(* PLC project OOP_Curso, Beckhoff Automation GmbH TwinCAT PLC Control 3.5.13.21 *)
(* stored: creationDateTime 2023-04-23T11:42:48.8573622, modificationDateTime 2023-04-23T11:42:48.8641947 *)

INTERFACE I_Employee
METHOD GetFullName : STRING
VAR_INPUT
END_VAR
END_METHOD
METHOD GetMonthlySalary : LREAL
VAR_INPUT
END_VAR
END_METHOD
PROPERTY nPersonnelNumber : UINT
END_PROPERTY
PROPERTY sFirstName : STRING
END_PROPERTY
PROPERTY sLastName : STRING
END_PROPERTY
END_INTERFACE

INTERFACE I_Employee_1
METHOD GetFullName : STRING
VAR_INPUT
END_VAR
END_METHOD
METHOD GetMonthlySalary : LREAL
VAR_INPUT
END_VAR
END_METHOD
PROPERTY nPersonnelNumber : UINT
END_PROPERTY
PROPERTY sFirstName : STRING
END_PROPERTY
PROPERTY sLastName : STRING
END_PROPERTY
END_INTERFACE

{attribute 'hide_all_locals'}
FUNCTION_BLOCK PUBLIC FB_ContractEmployee EXTENDS FB_Employee
VAR_INPUT
END_VAR
VAR_OUTPUT
END_VAR
VAR
	nHourlyPayBacking		:	UINT;
	nMonthlyHoursBacking	:	UINT;
END_VAR

            
          

METHOD PUBLIC GetMonthlySalary : LREAL
VAR_INPUT
END_VAR
                  GetMonthlySalary := nMonthlyHours * nHourlyPay;
                
END_METHOD

{attribute 'monitoring' := 'variable'}
PROPERTY PUBLIC nHourlyPay : UINT
GET
VAR
END_VAR
                    nHourlyPay := nHourlyPayBacking;
                  
END_GET
SET
VAR
END_VAR
                    nHourlyPayBacking := nHourlyPay;
                  
END_SET
END_PROPERTY

{attribute 'monitoring' := 'variable'}
PROPERTY PUBLIC nMonthlyHours : UINT
GET
VAR
END_VAR
                    nMonthlyHours := nMonthlyHoursBacking;
                  
END_GET
SET
VAR
END_VAR
                    nMonthlyHoursBacking := nMonthlyHours;
                  
END_SET
END_PROPERTY
END_FUNCTION_BLOCK

{attribute 'hide_all_locals'}
FUNCTION_BLOCK PUBLIC ABSTRACT FB_Employee
VAR_INPUT
END_VAR
VAR_OUTPUT
END_VAR
VAR
	nPersonnelNumberBacking :	UINT;
	sFirstNameBacking		:	STRING;
	sLastNameBacking		:	STRING;
END_VAR

            
          

METHOD PUBLIC GetFullName : STRING
VAR_INPUT
END_VAR
                  GetFullName := CONCAT(CONCAT(CONCAT(CONCAT(TO_STRING(nPersonnelNumber), ': '), sFirstName), ' '), sLastName);

                
END_METHOD

METHOD PUBLIC ABSTRACT GetMonthlySalary : LREAL
VAR_INPUT
END_VAR
                  
                
END_METHOD

{attribute 'monitoring' := 'variable'}
PROPERTY PUBLIC nPersonnelNumber : UINT
GET
VAR
END_VAR
                    nPersonnelNumber := nPersonnelNumberBacking;
                  
END_GET
SET
VAR
END_VAR
                    nPersonnelNumberBacking := nPersonnelNumber;
                  
END_SET
END_PROPERTY

{attribute 'monitoring' := 'variable'}
PROPERTY PUBLIC sFirstName : STRING
GET
VAR
END_VAR
                    sFirstName := sFirstNameBacking;
                  
END_GET
SET
VAR
END_VAR
                    sFirstNameBacking := sFirstName;
                  
END_SET
END_PROPERTY

{attribute 'monitoring' := 'variable'}
PROPERTY PUBLIC sLastName : STRING
GET
VAR
END_VAR
                    sLastName := sLastNameBacking;
                  
END_GET
SET
VAR
END_VAR
                    sLastNameBacking := sLastName;
                  
END_SET
END_PROPERTY
END_FUNCTION_BLOCK

{attribute 'hide_all_locals'}
FUNCTION_BLOCK PUBLIC FB_FullTimeEmployee EXTENDS FB_Employee
VAR_INPUT
END_VAR
VAR_OUTPUT
END_VAR
VAR
	nAnnualSalaryBacking	:	UINT;
END_VAR

            
          

METHOD PUBLIC GetMonthlySalary : LREAL
VAR_INPUT
END_VAR
                  GetMonthlySalary := nAnnualSalary / 12;
                
END_METHOD

{attribute 'monitoring' := 'variable'}
PROPERTY PUBLIC nAnnualSalary : UINT
GET
VAR
END_VAR
                    nAnnualSalary := nAnnualSalaryBacking;
                  
END_GET
SET
VAR
END_VAR
                    nAnnualSalaryBacking := nAnnualSalary;
                  
END_SET
END_PROPERTY
END_FUNCTION_BLOCK

PROGRAM POU_Main_FB_Abstract
VAR	
	fbFullTimeEmployee	:	FB_FullTimeEmployee;
	fbContractEmployee	:	FB_ContractEmployee;
	refEmployee			:	REFERENCE TO FB_Employee;
	aFullName			:	ARRAY[1..2] OF STRING;
	aMonthlySalary		:	ARRAY[1..2] OF LREAL;
END_VAR

            fbFullTimeEmployee.nPersonnelNumber := 1;
fbFullTimeEmployee.sFirstName := 'John';
fbFullTimeEmployee.sLastName := 'Taylor';
fbFullTimeEmployee.nAnnualSalary := 60000;
// access via concrete FB
aFullName[1] := fbFullTimeEmployee.GetFullName();
aMonthlySalary[1] := fbFullTimeEmployee.GetMonthlySalary();
// access via abstract FB
refEmployee REF= fbFullTimeEmployee;
aFullName[1] := refEmployee.GetFullName();
aMonthlySalary[1] := refEmployee.GetMonthlySalary();

fbContractEmployee.nPersonnelNumber := 2;
fbContractEmployee.sFirstName := 'Tim';
fbContractEmployee.sLastName := 'Brown';
fbContractEmployee.nMonthlyHours := 160;
fbContractEmployee.nHourlyPay := 35;
// access via concrete FB
aFullName[2] := fbContractEmployee.GetFullName();
aMonthlySalary[2] := fbContractEmployee.GetMonthlySalary();
// access via abstract FB
refEmployee REF= fbContractEmployee;
aFullName[2] := refEmployee.GetFullName();
aMonthlySalary[2] := refEmployee.GetMonthlySalary();
          
END_PROGRAM

{attribute 'hide_all_locals'}
FUNCTION_BLOCK PUBLIC FB_ContractEmployee_1 IMPLEMENTS I_Employee
VAR_INPUT
END_VAR
VAR_OUTPUT
END_VAR
VAR
	nPersonnelNumberBacking :	UINT;
	sFirstNameBacking		:	STRING;
	sLastNameBacking		:	STRING;
	
	nHourlyPayBacking		:	UINT;
	nMonthlyHoursBacking	:	UINT;
END_VAR

            
          

METHOD GetFullName : STRING
VAR_INPUT
END_VAR
                  GetFullName := CONCAT(CONCAT(CONCAT(CONCAT(TO_STRING(nPersonnelNumber), ': '), sFirstName), ' '), sLastName);
                
END_METHOD

METHOD PUBLIC GetMonthlySalary : LREAL
VAR_INPUT
END_VAR
                  GetMonthlySalary := nMonthlyHours * nHourlyPay;
                
END_METHOD

{attribute 'monitoring' := 'variable'}
PROPERTY PUBLIC nHourlyPay : UINT
GET
VAR
END_VAR
                    nHourlyPay := nHourlyPayBacking;
                  
END_GET
SET
VAR
END_VAR
                    nHourlyPayBacking := nHourlyPay;
                  
END_SET
END_PROPERTY

{attribute 'monitoring' := 'variable'}
PROPERTY PUBLIC nMonthlyHours : UINT
GET
VAR
END_VAR
                    nMonthlyHours := nMonthlyHoursBacking;
                  
END_GET
SET
VAR
END_VAR
                    nMonthlyHoursBacking := nMonthlyHours;
                  
END_SET
END_PROPERTY

{attribute 'monitoring' := 'variable'}
PROPERTY nPersonnelNumber : UINT
GET
VAR
END_VAR
                    nPersonnelNumber := nPersonnelNumberBacking;
                  
END_GET
SET
VAR
END_VAR
                    nPersonnelNumberBacking := nPersonnelNumber;
                  
END_SET
END_PROPERTY

{attribute 'monitoring' := 'variable'}
PROPERTY sFirstName : STRING
GET
VAR
END_VAR
                    sFirstName := sFirstNameBacking;
                  
END_GET
SET
VAR
END_VAR
                    sFirstNameBacking := sFirstName;
                  
END_SET
END_PROPERTY

{attribute 'monitoring' := 'variable'}
PROPERTY sLastName : STRING
GET
VAR
END_VAR
                    sLastName := sLastNameBacking;
                  
END_GET
SET
VAR
END_VAR
                    sLastNameBacking := sLastName;
                  
END_SET
END_PROPERTY
END_FUNCTION_BLOCK

{attribute 'hide_all_locals'}
FUNCTION_BLOCK PUBLIC FB_FullTimeEmployee_1 IMPLEMENTS I_Employee
VAR_INPUT
END_VAR
VAR_OUTPUT
END_VAR
VAR
	nPersonnelNumberBacking :	UINT;
	sFirstNameBacking		:	STRING;
	sLastNameBacking		:	STRING;	

	nAnnualSalaryBacking	:	UINT;
END_VAR

            
          

METHOD GetFullName : STRING
VAR_INPUT
END_VAR
                  GetFullName := CONCAT(CONCAT(CONCAT(CONCAT(TO_STRING(nPersonnelNumber), ': '), sFirstName), ' '), sLastName);
                
END_METHOD

METHOD PUBLIC GetMonthlySalary : LREAL
VAR_INPUT
END_VAR
                  GetMonthlySalary := nAnnualSalary / 12;
                
END_METHOD

{attribute 'monitoring' := 'variable'}
PROPERTY PUBLIC nAnnualSalary : UINT
GET
VAR
END_VAR
                    nAnnualSalary := nAnnualSalaryBacking;
                  
END_GET
SET
VAR
END_VAR
                    nAnnualSalaryBacking := nAnnualSalary;
                  
END_SET
END_PROPERTY

{attribute 'monitoring' := 'variable'}
PROPERTY nPersonnelNumber : UINT
GET
VAR
END_VAR
                    nPersonnelNumber := nPersonnelNumberBacking;
                  
END_GET
SET
VAR
END_VAR
                    nPersonnelNumberBacking := nPersonnelNumber;
                  
END_SET
END_PROPERTY

{attribute 'monitoring' := 'variable'}
PROPERTY sFirstName : STRING
GET
VAR
END_VAR
                    sFirstName := sFirstNameBacking;
                  
END_GET
SET
VAR
END_VAR
                    sFirstNameBacking := sFirstName;
                  
END_SET
END_PROPERTY

{attribute 'monitoring' := 'variable'}
PROPERTY sLastName : STRING
GET
VAR
END_VAR
                    sLastName := sLastNameBacking;
                  
END_GET
SET
VAR
END_VAR
                    sLastNameBacking := sLastName;
                  
END_SET
END_PROPERTY
END_FUNCTION_BLOCK

PROGRAM POU_Main_Interfaz
VAR
	fbFullTimeEmployee	:	FB_FullTimeEmployee_1;
	fbContractEmployee	:	FB_ContractEmployee_1;
	ipEmployee			:	I_Employee;
	aFullName			:	ARRAY[1..2] OF STRING;
	aMonthlySalary		:	ARRAY[1..2] OF LREAL;
END_VAR

            fbFullTimeEmployee.nPersonnelNumber := 1;
fbFullTimeEmployee.sFirstName := 'John';
fbFullTimeEmployee.sLastName := 'Taylor';
fbFullTimeEmployee.nAnnualSalary := 60000;
// access via FB
aFullName[1] := fbFullTimeEmployee.GetFullName();
aMonthlySalary[1] := fbFullTimeEmployee.GetMonthlySalary();
// access via interface
ipEmployee := fbFullTimeEmployee;
aFullName[1] := ipEmployee.GetFullName();
aMonthlySalary[1] := ipEmployee.GetMonthlySalary();

fbContractEmployee.nPersonnelNumber := 2;
fbContractEmployee.sFirstName := 'Tim';
fbContractEmployee.sLastName := 'Brown';
fbContractEmployee.nMonthlyHours := 160;
fbContractEmployee.nHourlyPay := 35;
// access via FB
aFullName[2] := fbContractEmployee.GetFullName();
aMonthlySalary[2] := fbContractEmployee.GetMonthlySalary();
// access via interface
ipEmployee := fbContractEmployee;
aFullName[2] := ipEmployee.GetFullName();
aMonthlySalary[2] := ipEmployee.GetMonthlySalary();
          
END_PROGRAM

{attribute 'hide_all_locals'}
FUNCTION_BLOCK PUBLIC FB_ContractEmployee_2 EXTENDS FB_Employee_1
VAR_INPUT
END_VAR
VAR_OUTPUT
END_VAR
VAR
	nHourlyPayBacking		:	UINT;
	nMonthlyHoursBacking	:	UINT;
END_VAR

            
          

METHOD PUBLIC GetMonthlySalary : LREAL
VAR_INPUT
END_VAR
                  GetMonthlySalary := nMonthlyHours * nHourlyPay;
                
END_METHOD

{attribute 'monitoring' := 'variable'}
PROPERTY PUBLIC nHourlyPay : UINT
GET
VAR
END_VAR
                    nHourlyPay := nHourlyPayBacking;
                  
END_GET
SET
VAR
END_VAR
                    nHourlyPayBacking := nHourlyPay;
                  
END_SET
END_PROPERTY

{attribute 'monitoring' := 'variable'}
PROPERTY PUBLIC nMonthlyHours : UINT
GET
VAR
END_VAR
                    nMonthlyHours := nMonthlyHoursBacking;
                  
END_GET
SET
VAR
END_VAR
                    nMonthlyHoursBacking := nMonthlyHours;
                  
END_SET
END_PROPERTY
END_FUNCTION_BLOCK

{attribute 'hide_all_locals'}
FUNCTION_BLOCK PUBLIC ABSTRACT FB_Employee_1 IMPLEMENTS I_Employee_1
VAR_INPUT
END_VAR
VAR_OUTPUT
END_VAR
VAR
	nPersonnelNumberBacking :	UINT;
	sFirstNameBacking		:	STRING;
	sLastNameBacking		:	STRING;
END_VAR

            
          

METHOD PUBLIC GetFullName : STRING
VAR_INPUT
END_VAR
                  GetFullName := CONCAT(CONCAT(CONCAT(CONCAT(TO_STRING(nPersonnelNumber), ': '), sFirstName), ' '), sLastName);

                
END_METHOD

METHOD PUBLIC ABSTRACT GetMonthlySalary : LREAL
VAR_INPUT
END_VAR
                  
                
END_METHOD

{attribute 'monitoring' := 'variable'}
PROPERTY PUBLIC nPersonnelNumber : UINT
GET
VAR
END_VAR
                    nPersonnelNumber := nPersonnelNumberBacking;
                  
END_GET
SET
VAR
END_VAR
                    nPersonnelNumberBacking := nPersonnelNumber;
                  
END_SET
END_PROPERTY

{attribute 'monitoring' := 'variable'}
PROPERTY PUBLIC sFirstName : STRING
GET
VAR
END_VAR
                    sFirstName := sFirstNameBacking;
                  
END_GET
SET
VAR
END_VAR
                    sFirstNameBacking := sFirstName;
                  
END_SET
END_PROPERTY

{attribute 'monitoring' := 'variable'}
PROPERTY PUBLIC sLastName : STRING
GET
VAR
END_VAR
                    sLastName := sLastNameBacking;
                  
END_GET
SET
VAR
END_VAR
                    sLastNameBacking := sLastName;
                  
END_SET
END_PROPERTY
END_FUNCTION_BLOCK

{attribute 'hide_all_locals'}
FUNCTION_BLOCK PUBLIC FB_FullTimeEmployee_2 EXTENDS FB_Employee_1
VAR_INPUT
END_VAR
VAR_OUTPUT
END_VAR
VAR
	nAnnualSalaryBacking	:	UINT;
END_VAR

            
          

METHOD PUBLIC GetMonthlySalary : LREAL
VAR_INPUT
END_VAR
                  GetMonthlySalary := nAnnualSalary / 12;
                
END_METHOD

{attribute 'monitoring' := 'variable'}
PROPERTY PUBLIC nAnnualSalary : UINT
GET
VAR
END_VAR
                    nAnnualSalary := nAnnualSalaryBacking;
                  
END_GET
SET
VAR
END_VAR
                    nAnnualSalaryBacking := nAnnualSalary;
                  
END_SET
END_PROPERTY
END_FUNCTION_BLOCK

PROGRAM POU_Main_Combinacion
VAR
	fbFullTimeEmployee	:	FB_FullTimeEmployee_2;
	fbContractEmployee	:	FB_ContractEmployee_2;
	refEmployee			:	REFERENCE TO FB_Employee_1;
	ipEmployee			:	I_Employee_1;	
	aFullName			:	ARRAY[1..2] OF STRING;
	aMonthlySalary		:	ARRAY[1..2] OF LREAL;
END_VAR

            fbFullTimeEmployee.nPersonnelNumber := 1;
fbFullTimeEmployee.sFirstName := 'John';
fbFullTimeEmployee.sLastName := 'Taylor';
fbFullTimeEmployee.nAnnualSalary := 60000;
// access via concrete FB
aFullName[1] := fbFullTimeEmployee.GetFullName();
aMonthlySalary[1] := fbFullTimeEmployee.GetMonthlySalary();
// access via abstract FB
refEmployee REF= fbFullTimeEmployee;
aFullName[1] := refEmployee.GetFullName();
aMonthlySalary[1] := refEmployee.GetMonthlySalary();
// access via interface
ipEmployee := fbFullTimeEmployee;
aFullName[1] := ipEmployee.GetFullName();
aMonthlySalary[1] := ipEmployee.GetMonthlySalary();

fbContractEmployee.nPersonnelNumber := 2;
fbContractEmployee.sFirstName := 'Tim';
fbContractEmployee.sLastName := 'Brown';
fbContractEmployee.nMonthlyHours := 160;
fbContractEmployee.nHourlyPay := 35;
// access via concrete FB
aFullName[2] := fbContractEmployee.GetFullName();
aMonthlySalary[2] := fbContractEmployee.GetMonthlySalary();
// access via abstract FB
refEmployee REF= fbContractEmployee;
aFullName[2] := refEmployee.GetFullName();
aMonthlySalary[2] := refEmployee.GetMonthlySalary();
// access via interface
ipEmployee := fbContractEmployee;
aFullName[2] := ipEmployee.GetFullName();
aMonthlySalary[2] := ipEmployee.GetMonthlySalary();
          
END_PROGRAM
